FUNCTION_BLOCK Conveyor1Controller (* Controller of Conveyor 1 *)
  (* Standard: 61499-2 *)
  (* Version 0.3, 2009-09-15, JHC, Holobloc Inc, Changed transition priorities. *)
  (* Version 0.2, 2003-12-04, JHC, Rockwell Automation, Renamed for better indexing. *)
  (* Version 0.1, 2002-11-05, JHC, Rockwell Automation, Corrected missing ST element in Algorithm REQ. *)
  (* Version 0.0, 2000-05-30, JHC, Rockwell Automation *)
  (* Compiler header: package fb.rt.dasdA1.A2.Conveyor1; *)
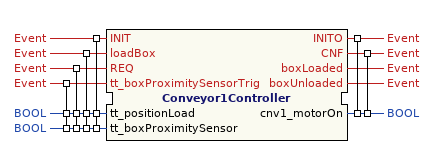
  EVENT_INPUT
    INIT WITH tt_positionLoad, tt_boxProximitySensor; (* Initialization Request *)
    loadBox WITH tt_boxProximitySensor, tt_positionLoad;
    REQ WITH tt_positionLoad, tt_boxProximitySensor;
    tt_boxProximitySensorTrig WITH tt_positionLoad, tt_boxProximitySensor;
  END_EVENT
  EVENT_OUTPUT
    INITO WITH cnv1_motorOn; (* Initialization Confirm *)
    CNF WITH cnv1_motorOn; (* Execution Confirmation *)
    boxLoaded;
    boxUnloaded;
  END_EVENT
  VAR_INPUT
    tt_positionLoad : BOOL;
    tt_boxProximitySensor : BOOL;
  END_VAR
  VAR_OUTPUT
    cnv1_motorOn : BOOL;
  END_VAR
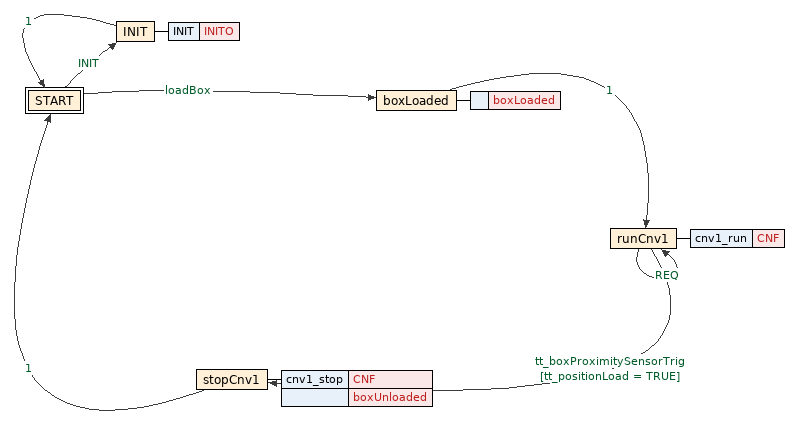
  EC_STATES
    START; (* Initial State *)
    INIT : INIT -> INITO; (* Initialization *)
    runCnv1 : cnv1_run -> CNF;
    stopCnv1 : cnv1_stop -> CNF, -> boxUnloaded;
    boxLoaded : -> boxLoaded;
  END_STATES
  EC_TRANSITIONS
    INIT TO START := 1;
    START TO INIT := INIT;
    runCnv1 TO stopCnv1 := tt_boxProximitySensorTrig [tt_positionLoad = TRUE];
    stopCnv1 TO START := 1;
    runCnv1 TO runCnv1 := REQ;
    START TO boxLoaded := loadBox;
    boxLoaded TO runCnv1 := 1;
  END_TRANSITIONS
  ALGORITHM INIT IN ST: (* Initialization algorithm *)
// tt_positionLoad := FALSE;
// tt_boxProximitySensor := FALSE;
cnv1_motorOn := FALSE;
  END_ALGORITHM
  ALGORITHM cnv1_run IN ST:
// Control the motor depending of states of the
// turn table´s box proximity sensor and turn table´s
// position
IF tt_boxProximitySensor = FALSE
	AND tt_positionLoad = TRUE
THEN
	cnv1_motorOn := TRUE;
ELSE
	cnv1_motorOn := FALSE;
END_IF;
  END_ALGORITHM
  ALGORITHM cnv1_stop IN ST:
cnv1_motorOn := FALSE;
  END_ALGORITHM
END_FUNCTION_BLOCK
